{attribute 'GeneratedUsingTerminal: EL3182-0000-0016'}
{attribute addProperty BoxType "EL3182-0000-0016"}
{attribute addProperty Id "Ch_1_Al_InputsCh_1_Al_Inputs_4794C08310"}
{attribute addProperty CRC "2717575001"}
{attribute addProperty Size "10"}
TYPE Ch_1_A1FAE759 :
STRUCT
	{attribute addProperty Name "Ch_1_Al_Inputs"}
	Ch_1_Al_Inputs  : Ch_1_Al_Inputs_4794C083;
END_STRUCT
END_TYPE

(* stored: Version 1.2.0.0, ProductVersion 3.1.4024.11
   DUT Ch_1_A1FAE759: Id {d45aecfb-a26d-4c8c-89cb-a593c9831366} *)
